Fanuc KAREL source: port_UIN.kl

PROGRAM TP
%NOLOCKGROUP
VAR
 x: BOOLEAN
BEGIN
 x = UIN[3]
END TP
